// TwinCAT 3 PLC project PlcTemplateTests
// Title: PlcTemplateTests
// Company: Vortex.Library
// ProjectVersion: 0.6.0.913
// ProgramVersion: 3.1.4024.12
// libraries:
//   PlcTemplate, 0.6.0.913 (Vortex.Library)
//   Tc2_Standard, * (Beckhoff Automation GmbH)
//   Tc2_System, * (Beckhoff Automation GmbH)
//   Tc3_Module, * (Beckhoff Automation GmbH)
//   TcoCore, 0.6.0.913 (Vortex.Library)
// project tree:
//   / PlcTask.TcTTO (not stored)
//   POUs/ MAIN.TcPOU, SampleComponentTests.TcPOU
// (motion and I/O tree: see PLC project plctemplate)
// real-time tasks:
//   TASK PlcTask: cycle T#10ms, priority 20, ADS port 350
//   TASK PlcTask1: cycle T#10ms, priority 21, ADS port 351

// ---- POUs/MAIN.TcPOU
PROGRAM MAIN
VAR
    _sampleComponentTests : SampleComponentTests;
END_VAR

END_PROGRAM

// ---- POUs/SampleComponentTests.TcPOU
FUNCTION_BLOCK SampleComponentTests EXTENDS _internals_TcoContext
VAR
    _sut : PlcTemplate.SampleComponent(THIS^);
END_VAR

{attribute 'TcRpcEnable'}
METHOD INTERNAL AddTwoNumbersTest : INT
VAR_INPUT
    NumberOne : INT;
    NumberTwo : INT;
END_VAR
AddTwoNumbersTest := _sut.AddTwoNumbers(NumberOne, NumberTwo);
END_METHOD

METHOD PROTECTED Main
END_METHOD

{attribute 'TcRpcEnable'}
METHOD INTERNAL WaitForModuloTest : BOOL
VAR_INPUT
    Modulo : INT;
END_VAR
WaitForModuloTest := _sut.WaitForModulo(Modulo);
END_METHOD

END_FUNCTION_BLOCK
